{attribute 'qualified_only'}
{attribute 'strict'}
TYPE E_CommandResultCode :
(
	Init := 0,
	Running := 1,
	Done := 2,
	Cancelled := 3
) UINT;
END_TYPE

(* stored: Version 1.1.0.1, ProductVersion 3.1.4022.10
   DUT E_CommandResultCode: Id {86e90a2a-1bfd-4ab0-9e94-fea458698174} *)
